SUBAPPLICATION Uebung_160 (* Motor Links/Rechtslauf *)
  (* Standard: 61499-2; Description: Copyright (c) 2023 Meisterschulen am Ostbahnhof This program and the accompanying materials are made available under the terms of the Eclipse Public License 2.0 which is available at https://www.eclipse.org/legal/epl-2.0/ SPDX-License-Identifier: EPL-2.0 *)
  (* Version 1.0, 2023-10-23, Franz Höpfinger, Meisterschulen am Ostbahnhof *)
  PACKAGE Uebungen;
  IMPORT logiBUS::io::DI::logiBUS_DI::Input_I1;
  IMPORT logiBUS::io::DI::logiBUS_DI::Input_I2;
  IMPORT logiBUS::io::DQ::logiBUS_DO::Output_Q5;
  IMPORT logiBUS::io::DQ::logiBUS_DO::Output_Q56;
  IMPORT logiBUS::io::DQ::logiBUS_DO::Output_Q6;
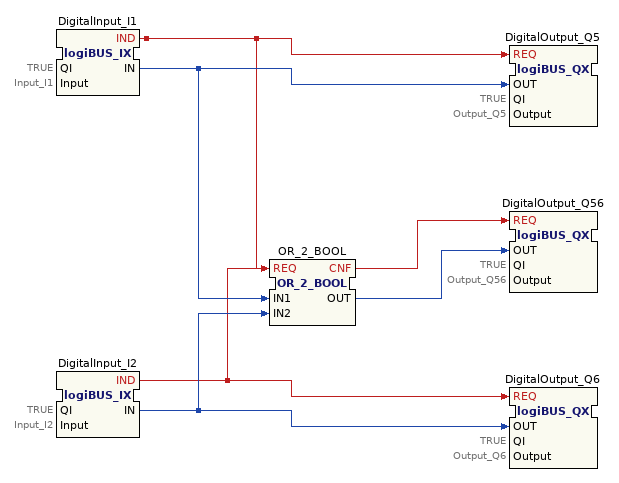
  FBS
    DigitalOutput_Q6 : logiBUS::io::DQ::logiBUS_QX(QI := TRUE, Output := Output_Q6);
    DigitalInput_I2 : logiBUS::io::DI::logiBUS_IX(QI := TRUE, Input := Input_I2);
    OR_2_BOOL : iec61131::bitwiseOperators::OR_2_BOOL;
    DigitalInput_I1 : logiBUS::io::DI::logiBUS_IX(QI := TRUE, Input := Input_I1);
    DigitalOutput_Q5 : logiBUS::io::DQ::logiBUS_QX(QI := TRUE, Output := Output_Q5);
    DigitalOutput_Q56 : logiBUS::io::DQ::logiBUS_QX(QI := TRUE, Output := Output_Q56);
  END_FBS
  EVENT_CONNECTIONS
    DigitalInput_I2.IND TO DigitalOutput_Q6.REQ;
    DigitalInput_I1.IND TO DigitalOutput_Q5.REQ;
    OR_2_BOOL.CNF TO DigitalOutput_Q56.REQ;
    DigitalInput_I2.IND TO OR_2_BOOL.REQ;
    DigitalInput_I1.IND TO OR_2_BOOL.REQ;
  END_CONNECTIONS
  DATA_CONNECTIONS
    DigitalInput_I2.IN TO DigitalOutput_Q6.OUT;
    DigitalInput_I1.IN TO DigitalOutput_Q5.OUT;
    OR_2_BOOL.OUT TO DigitalOutput_Q56.OUT;
    DigitalInput_I1.IN TO OR_2_BOOL.IN1;
    DigitalInput_I2.IN TO OR_2_BOOL.IN2;
  END_CONNECTIONS
END_SUBAPPLICATION
